Fanuc KAREL source: kd00014.KL

-- PROVISIONAL review KL for V1013-1; original PC SHA256 100f1b2e6710e144bb8e7b1267c8997fd03567316835a5a82d583712cc41e61e
-- Incomplete behavior may be omitted. Consult companion uncertainty JSON. Do not deploy.
PROGRAM KD00014
%NOLOCKGROUP
VAR
  I : INTEGER
  J : INTEGER
  B : BOOLEAN
  R : REAL
  S : STRING[80]
BEGIN
  -- UNRESOLVED_PC offsets 5-9; opcodes 9C,9D,1A
  -- UNRESOLVED_PC offsets 14-18; opcodes 7F
END KD00014
